{attribute 'linkalways'} 
{attribute 'no_explicit_call' := 'This FB is a CLASS and must be accessed using methods or properties'}
{attribute 'enable_dynamic_creation'}
FUNCTION_BLOCK _BYTE EXTENDS NumericDatatypeBase
VAR
	localData : BYTE;
	activeData : REFERENCE TO BYTE REF= localData;
END_VAR

PROPERTY PUBLIC Address : PVOID
GET
Address := ADR(activeData);
END_GET
END_PROPERTY

METHOD PUBLIC ClearReference
VAR_INPUT
END_VAR
activeData REF= localData;
END_METHOD

METHOD PUBLIC Clone : I_Datatype
VAR
    pClone : POINTER TO _BYTE;
END_VAR
pClone := __NEW(_BYTE(InitialValue := Value));
Clone := pClone^;
END_METHOD

METHOD FB_init : BOOL
VAR_INPUT
	bInitRetains : BOOL; // if TRUE, the retain variables are initialized (warm start / cold start)
	bInCopyCode : BOOL;  // if TRUE, the instance afterwards gets moved into the copy code (online change)
	InitialValue : BYTE;
END_VAR
localData := InitialValue;
END_METHOD

PROPERTY PUBLIC IsFloat : BOOL
GET
IsFloat := FALSE;
END_GET
END_PROPERTY

PROPERTY PUBLIC IsSigned : BOOL
GET
IsSigned := FALSE;
END_GET
END_PROPERTY

METHOD PUBLIC MakeReferenceTo
VAR_INPUT
	ReferenceTarget : REFERENCE TO BYTE;
END_VAR
activeData REF= ReferenceTarget;
END_METHOD

PROPERTY PUBLIC MaxValue : BYTE
GET
MaxValue := DatatypeLimits.BYTE_MAX_VALUE;
END_GET
END_PROPERTY

PROPERTY PUBLIC MinValue : BYTE
GET
MinValue := DatatypeLimits.BYTE_MIN_VALUE;
END_GET
END_PROPERTY

METHOD PROTECTED SerializeMaxValue
VAR_INPUT
	Serializer : I_Serializer;
END_VAR
Serializer.AddByte(MaxValue);
END_METHOD

METHOD PROTECTED SerializeMinValue
VAR_INPUT
	Serializer : I_Serializer;
END_VAR
Serializer.AddByte(MinValue);
END_METHOD

METHOD PUBLIC SerializeWith
VAR_INPUT
	Serializer : I_Serializer;
END_VAR
Serializer.AddByte(activeData);
END_METHOD

PROPERTY PUBLIC Size : UDINT
GET
Size := SIZEOF(activeData);
END_GET
END_PROPERTY

METHOD TryDeserializeFrom : BOOL
VAR_INPUT
	Deserializer : I_Deserializer;
	Feedback : I_DeserializerFeedback;
END_VAR
TryDeserializeFrom := Deserializer.TryGetByte(activeData, Feedback);
END_METHOD

METHOD TryMakeReferenceTo : BOOL
VAR_INPUT
	Target : I_Datatype;
END_VAR
VAR
	pTargetData : POINTER TO BYTE;
END_VAR
IF NOT (Target.TypeName = TypeName) THEN
	RETURN;
END_IF

pTargetData := Target.Address;
activeData REF= pTargetData^;
TryMakeReferenceTo := TRUE;
END_METHOD

PROPERTY PUBLIC TypeName : T_MAXSTRING
GET
TypeName := 'BYTE';
END_GET
END_PROPERTY

PROPERTY PUBLIC Value : REFERENCE TO BYTE
GET
Value REF= activeData;
END_GET
END_PROPERTY

END_FUNCTION_BLOCK

(* stored: Version 1.1.0.1, ProductVersion 3.1.4024.12
   POU _BYTE: Id {a9dbf698-1a18-4707-9ef0-fbce4f618e11}, SpecialFunc None
   Folder Constructor: Id {fa267d6b-8c7b-4359-96c0-f02cc7b932d0}
   Folder Protected: Id {222d1d66-3f7c-4985-b740-ce79b05436e8}
   Property Address: Id {5ce19b2d-651a-4a25-b6a6-01ff899db0f8}
   Get Get: Id {7fd7f58b-6979-493e-acb5-d7793cd419f7}
   Method ClearReference: Id {90d0cb8d-9d75-42bb-97a2-194d3ec9ef48}
   Method Clone: Id {4a9ce530-ba07-4c4e-abe4-c2653dedf808}
   Method FB_init: Id {6fbb58fb-f044-4a43-b1fb-69a7f8f9d613}
   Property IsFloat: Id {cd361d45-fab1-41c3-bbeb-9ece597102c0}
   Get Get: Id {404e6ad1-06a2-487f-9cd1-6593de0de060}
   Property IsSigned: Id {2b27a8d2-32c8-40fb-90a3-f889753605dc}
   Get Get: Id {7eed14a3-f39f-44ac-9079-82ded48e156d}
   Method MakeReferenceTo: Id {b0685fb2-a91a-4300-abc8-88a12c9d7e72}
   Property MaxValue: Id {ef5acad3-9437-4bee-a7d9-d491426c23a8}
   Get Get: Id {161349e0-ee00-42fe-b878-d6ca1c341b16}
   Property MinValue: Id {1821b4a8-b9b9-401c-a653-702ea2fe4b74}
   Get Get: Id {23b184e0-a6b1-4e76-a981-a37469b5ac76}
   Method SerializeMaxValue: Id {83a9c987-f9fa-4e59-abc5-8ed3d4b66a51}
   Method SerializeMinValue: Id {c354d1f7-5954-4ef9-9175-fbcb9d1d79e4}
   Method SerializeWith: Id {ce7f0d95-b96d-4130-9347-86b3b9e7c3df}
   Property Size: Id {d7112066-4da8-4ba8-822f-a21d4ca31848}
   Get Get: Id {ba093846-e4ca-4d02-96d9-7a2a9207c9c2}
   Method TryDeserializeFrom: Id {45e1527e-5fd5-488f-b4e1-545ff415e63d}
   Method TryMakeReferenceTo: Id {74f83ec6-128b-4ae6-8a73-f5b688f705b6}
   Property TypeName: Id {b4983b3c-2ec5-456c-b6d1-9525ac82dec7}
   Get Get: Id {87bed962-fde5-4566-aea6-78880871f00b}
   Property Value: Id {869052aa-ea48-4c1b-8a92-2d71f2b07c0c}
   Get Get: Id {eb06258b-6ad4-49ce-a837-d23e7b145495} *)
